PROGRAM POU_NCI
VAR
	fb_BuildGroup: CfgBuild3DGroup;
	fb_ReconfigGroup: CfgReconfigGroup;
	fb_LoadProg: ItpLoadProgEx;
	fb_StartStop: ItpStartStopEx;
	fb_Reset: ItpResetEx2;
	
END_VAR

fb_BuildGroup(
	bExecute:= gcode.bBuildGroup, 
	nGroupId:= GVL.ChannelInput.GrpId, 
	nXAxisId:= GVL.As_Xa.NcToPlc.AxisId, 
	nYAxisId:= GVL.As_Y.NcToPlc.AxisId, 
	nZAxisId:= GVL.As_Z.NcToPlc.AxisId, 
	tTimeOut:= T#1S );
	
fb_ReconfigGroup(
	bExecute:= NOT(gcode.bBuildGroup), 
	nGroupId:= GVL.ChannelInput.GrpId, 
	tTimeOut:= T#1S );
	
ItpSetOverridePercent(fOverridePercent:= 100, sPlcToNci:= GVL.ChannelOutput);

fb_LoadProg(
	sNciToPlc:= GVL.ChannelInput, 
	bExecute:= gcode.bLoad, 
	sPrg:= '\HARD DISK\TWINCAT\Mc\Nci\Gcode_test1.nc', 
	nLength:= LEN('\HARD DISK\TWINCAT\Mc\Nci\Gcode_test1.nc'), 
	tTimeOut:= T#1S );
	
fb_StartStop(
	bStart:= gcode.bStart, 
	bStop:= gcode.bStop OR gvl.StopALL, 
	tTimeOut:= T#1S, 
	sNciToPlc:= GVL.ChannelInput );
	
fb_Reset(
	bExecute:= gcode.bReset, 
	tTimeOut:= T#1S, 
	sNciToPlc:= GVL.ChannelInput );

END_PROGRAM

(* stored: Version 1.1.0.1, ProductVersion 3.1.4024.2
   POU POU_NCI: Id {9c84d0cd-cbbc-4c86-9c9d-2561bd9b238b}, SpecialFunc None *)
